FUNCTION_BLOCK CounterBFB
  (* Standard: 61499-2 *)
  (* Version 0.1, 2016-00-15, Hammond, HAMMONDSDESKTOP *)
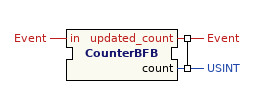
  EVENT_INPUT
    in;
  END_EVENT
  EVENT_OUTPUT
    updated_count WITH count;
  END_EVENT
  VAR_OUTPUT
    count : USINT := 10;
  END_VAR
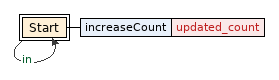
  EC_STATES
    Start : increaseCount -> updated_count;
  END_STATES
  EC_TRANSITIONS
    Start TO Start := in;
  END_TRANSITIONS
  ALGORITHM increaseCount IN C:
me->count++;
  END_ALGORITHM
END_FUNCTION_BLOCK
